FUNCTION_BLOCK FB_Labeler
VAR_INPUT
    nLabels : UDINT;
    pRoll   : POINTER TO UDINT;     // remaining labels on the roll, from the HMI
END_VAR
VAR_OUTPUT
    nRollsUsed : UDINT;
    bRollLow   : BOOL;
END_VAR
VAR CONSTANT
    cLabelsPerRoll : UDINT := 2000;
END_VAR

nRollsUsed := nLabels / cLabelsPerRoll;
IF pRoll <> 0 THEN
    bRollLow := pRoll^ < 100;
END_IF

END_FUNCTION_BLOCK

(* stored: Version 1.1.0.1, ProductVersion 3.1.4024.0
   POU FB_Labeler: Id {5a440053-e5a6-4ae4-853e-d3bc8412c14d}, SpecialFunc None *)
